Staubli VAL3: CloseFile.pgx

public program CloseFile(num x_nFileID (dimensions=1))
begin

  //文件标志符


  if x_nFileID<0 or x_nFileID>9
    return
  endIf

  //
  switch x_nFileID
    case 0
      $fileClose(0)
    break

    case 1
      $fileClose(1)
    break

    case 2
      $fileClose(2)
    break

    case 3
      $fileClose(3)
    break

    case 4
      $fileClose(4)
    break

    case 5
      $fileClose(5)
    break
    case 6
      $fileClose(6)
    break

    case 7
      $fileClose(7)
    break
    case 8
      $fileClose(8)
    break

    case 9
      $fileClose(9)
    break


  endSwitch


end
